VAR_GLOBAL

	stCamera								: ST_Camera;
	stLeakTesters							: ST_LeakTester;	
	stLSS									: ST_LSS;
	stProcessCylinder						: ST_ProcessCylinder;
	stProcessDoor							: ST_ProcessDoor;
	stVacuumCylinder						: ST_VacuumCylinder;

	stPuckLocker 							: ST_PuckLocker;
	
END_VAR

(* stored: Version 1.1.0.1, ProductVersion 3.1.4026.18
   GVL GVL_Stations: Id {51987edd-ecbc-463a-bda0-55117182c9fa} *)
